{attribute addProperty BoxType "ER3184-0002-0019"}
{attribute addProperty Id "AI_Standard_ChannelAT %I*ARRAY[0..3] OF AI_Standard_Channel_904746A2128160WcStateAT %I*WcState_F855686C1620InfoDataAT %I*InfoData_BC63D37F80100"}
{attribute addProperty CRC "975291572"}
{attribute addProperty SizeInBites "224"}
{attribute addProperty SizeInBytes "28"}
TYPE ER3184_55F04E99 :
STRUCT
	{attribute addProperty Name "AI_Standard_Channel"}
	AI_Standard_Channel : ARRAY[0..3] OF AI_Standard_Channel_904746A2;
	{attribute addProperty Name "WcState"}
	WcState : WcState_F855686C;
	{attribute addProperty Name "InfoData"}
	InfoData : InfoData_BC63D37F;
END_STRUCT
END_TYPE

(* stored: Version 1.2.0.0, ProductVersion 3.1.4024.9
   DUT ER3184_55F04E99: Id {c0f9bfa0-1a02-4e55-9530-6bccd90e5087} *)
